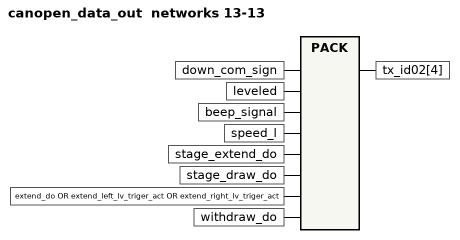
[picture p96: canopen_data_out (FBD) networks 13-13]
_FBD_ (* Function Block Diagram *)
NETWORK 1
	PACK(front_left_urt_ex_check, front_right_urt_ex_check, back_left_urt_ex_check, back_right_urt_ex_check, front_left_urt_drb_check, front_right_urt_drb_check, back_left_urt_drb_check, back_right_urt_drb_check) => tx_id01[0]
NETWORK 2
	PACK(front_left_Lv_ex_check, front_right_Lv_ex_check, back_left_Lv_ex_check, back_right_Lv_ex_check, front_left_Lv_drb_check, front_right_Lv_drb_check, back_left_Lv_drb_check, back_right_Lv_drb_check) => tx_id01[1]
NETWORK 3
	PACK(engine_run, engine_stop, accelerate_sb, decelerate_sb, down_force, tt_forcexx, standby_pump_check, water_pump_run_sb) => tx_id01[2]
NETWORK 4
	PACK(auto_manu_choice, left_side_choice, right_side_choice, level_extend_triger_left, level_extend_triger_right, auto_extend_triger_left OR auto_extend_triger_right, auto_drawback_triger_left OR auto_drawback_triger_right, remote_switch_leg) => tx_id01[3]
NETWORK 5
	PACK(FALSE, FALSE, FALSE, FALSE, FALSE, FALSE, FALSE, FALSE) => tx_id01[4]
NETWORK 6
	PACK(FALSE, FALSE, FALSE, FALSE, FALSE, FALSE, FALSE, FALSE) => tx_id01[5]
NETWORK 7
	PACK(arm_to_station, water_pump_check, left_groud_check1, left_groud_check2, oil_pump_check, FALSE, FALSE, FALSE) => tx_id01[6]
NETWORK 8
	PACK(FALSE, FALSE, FALSE, FALSE, FALSE, FALSE, FALSE, FALSE) => tx_id01[7]
NETWORK 9
	PACK(left_front_lv_ex_valve, right_front_lv_ex_valve, left_back_lv_ex_valve, right_back_lv_ex_valve, left_front_lv_drb_valve, right_front_lv_drb_valve, left_back_lv_drb_valve, right_back_lv_drb_valve) => tx_id02[0]
NETWORK 10
	PACK(enginer_run_ctl, enginer_stop_ctl, enginer_acc_ctl, enginer_dec_ctl, water_pump_ctl, up_valve_ctl, down_valve_ctl, over_level_sign) => tx_id02[1]
NETWORK 11
	PACK(triger_left_grd_sign, under_reset_ctl, standby_oil_pump, triger_flash, triger_no_drawback_sign, leveled_sign, alarmer_horn, FALSE) => tx_id02[2]
NETWORK 12
	PACK(FALSE, FALSE, FALSE, FALSE, FALSE, FALSE, FALSE, FALSE) => tx_id02[3]
NETWORK 13
	PACK(down_com_sign, leveled, beep_signal, speed_l, stage_extend_do, stage_draw_do, extend_do OR extend_left_lv_triger_act OR extend_right_lv_triger_act, withdraw_do) => tx_id02[4]
_END_FBD_
(* the same logic as Structured Text *)
(* Network 1 *)
tx_id01[0] := PACK(front_left_urt_ex_check, front_right_urt_ex_check, back_left_urt_ex_check, back_right_urt_ex_check, front_left_urt_drb_check, front_right_urt_drb_check, back_left_urt_drb_check, back_right_urt_drb_check);
(* Network 2 *)
tx_id01[1] := PACK(front_left_Lv_ex_check, front_right_Lv_ex_check, back_left_Lv_ex_check, back_right_Lv_ex_check, front_left_Lv_drb_check, front_right_Lv_drb_check, back_left_Lv_drb_check, back_right_Lv_drb_check);
(* Network 3 *)
tx_id01[2] := PACK(engine_run, engine_stop, accelerate_sb, decelerate_sb, down_force, tt_forcexx, standby_pump_check, water_pump_run_sb);
(* Network 4 *)
tx_id01[3] := PACK(auto_manu_choice, left_side_choice, right_side_choice, level_extend_triger_left, level_extend_triger_right, auto_extend_triger_left OR auto_extend_triger_right, auto_drawback_triger_left OR auto_drawback_triger_right, remote_switch_leg);
(* Network 5 *)
tx_id01[4] := PACK(FALSE, FALSE, FALSE, FALSE, FALSE, FALSE, FALSE, FALSE);
(* Network 6 *)
tx_id01[5] := PACK(FALSE, FALSE, FALSE, FALSE, FALSE, FALSE, FALSE, FALSE);
(* Network 7 *)
tx_id01[6] := PACK(arm_to_station, water_pump_check, left_groud_check1, left_groud_check2, oil_pump_check, FALSE, FALSE, FALSE);
(* Network 8 *)
tx_id01[7] := PACK(FALSE, FALSE, FALSE, FALSE, FALSE, FALSE, FALSE, FALSE);
(* Network 9 *)
tx_id02[0] := PACK(left_front_lv_ex_valve, right_front_lv_ex_valve, left_back_lv_ex_valve, right_back_lv_ex_valve, left_front_lv_drb_valve, right_front_lv_drb_valve, left_back_lv_drb_valve, right_back_lv_drb_valve);
(* Network 10 *)
tx_id02[1] := PACK(enginer_run_ctl, enginer_stop_ctl, enginer_acc_ctl, enginer_dec_ctl, water_pump_ctl, up_valve_ctl, down_valve_ctl, over_level_sign);
(* Network 11 *)
tx_id02[2] := PACK(triger_left_grd_sign, under_reset_ctl, standby_oil_pump, triger_flash, triger_no_drawback_sign, leveled_sign, alarmer_horn, FALSE);
(* Network 12 *)
tx_id02[3] := PACK(FALSE, FALSE, FALSE, FALSE, FALSE, FALSE, FALSE, FALSE);
(* Network 13 *)
tx_id02[4] := PACK(down_com_sign, leveled, beep_signal, speed_l, stage_extend_do, stage_draw_do, extend_do OR extend_left_lv_triger_act OR extend_right_lv_triger_act, withdraw_do);
END_PROGRAM

(* POU CANOPEN_DATA/digit_data_in, FBD *)
PROGRAM digit_data_in
VAR

	UNPACK1		: UNPACK;
	UNPACK2		: UNPACK;
	UNPACK3		: UNPACK;
	UNPACK4		: UNPACK;
	UNPACK5		: UNPACK;
	UNPACK6		: UNPACK;
	UNPACK7		: UNPACK;
	UNPACK8		: UNPACK;
	UNPACK9		: UNPACK;
	UNPACK10	: UNPACK;
	UNPACK11	: UNPACK;

END_VAR
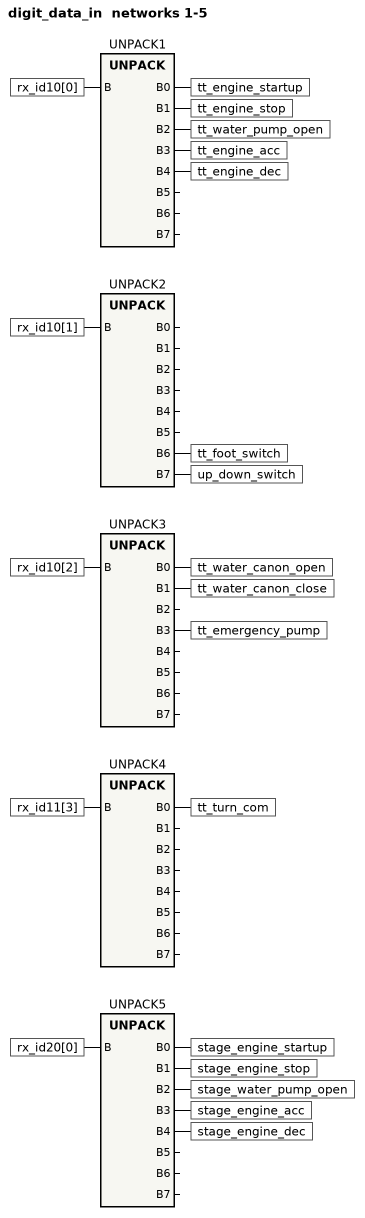
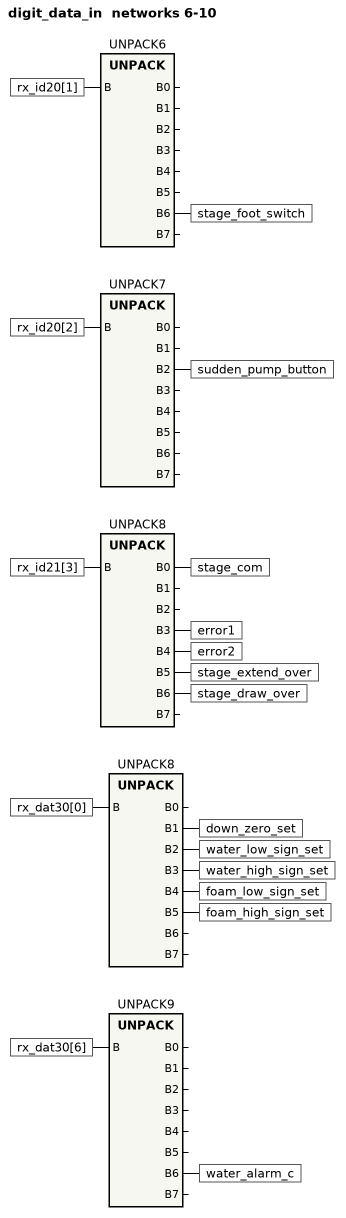
_FBD_ (* Function Block Diagram *)
NETWORK 1
	UNPACK1:UNPACK(B: rx_id10[0], B1 => tt_engine_stop, B2 => tt_water_pump_open, B3 => tt_engine_acc, B4 => tt_engine_dec) => tt_engine_startup
NETWORK 2
	UNPACK2:UNPACK(B: rx_id10[1], B6 => tt_foot_switch, B7 => up_down_switch)
NETWORK 3
	UNPACK3:UNPACK(B: rx_id10[2], B1 => tt_water_canon_close, B3 => tt_emergency_pump) => tt_water_canon_open
NETWORK 4
	UNPACK4:UNPACK(B: rx_id11[3]) => tt_turn_com
NETWORK 5
	UNPACK5:UNPACK(B: rx_id20[0], B1 => stage_engine_stop, B2 => stage_water_pump_open, B3 => stage_engine_acc, B4 => stage_engine_dec) => stage_engine_startup
NETWORK 6
	UNPACK6:UNPACK(B: rx_id20[1], B6 => stage_foot_switch)
NETWORK 7
	UNPACK7:UNPACK(B: rx_id20[2], B2 => sudden_pump_button)
NETWORK 8
	UNPACK8:UNPACK(B: rx_id21[3], B3 => error1, B4 => error2, B5 => stage_extend_over, B6 => stage_draw_over) => stage_com
NETWORK 9
	UNPACK8:UNPACK(B: rx_dat30[0], B1 => down_zero_set, B2 => water_low_sign_set, B3 => water_high_sign_set, B4 => foam_low_sign_set, B5 => foam_high_sign_set)
NETWORK 10
	UNPACK9:UNPACK(B: rx_dat30[6], B6 => water_alarm_c)
_END_FBD_
(* the same logic as Structured Text *)
(* Network 1 *)
UNPACK1(B := rx_id10[0]);
tt_engine_stop := UNPACK1.B1;
tt_water_pump_open := UNPACK1.B2;
tt_engine_acc := UNPACK1.B3;
tt_engine_dec := UNPACK1.B4;
tt_engine_startup := UNPACK1.B0;
(* Network 2 *)
UNPACK2(B := rx_id10[1]);
tt_foot_switch := UNPACK2.B6;
up_down_switch := UNPACK2.B7;
(* Network 3 *)
UNPACK3(B := rx_id10[2]);
tt_water_canon_close := UNPACK3.B1;
tt_emergency_pump := UNPACK3.B3;
tt_water_canon_open := UNPACK3.B0;
(* Network 4 *)
UNPACK4(B := rx_id11[3]);
tt_turn_com := UNPACK4.B0;
(* Network 5 *)
UNPACK5(B := rx_id20[0]);
stage_engine_stop := UNPACK5.B1;
stage_water_pump_open := UNPACK5.B2;
stage_engine_acc := UNPACK5.B3;
stage_engine_dec := UNPACK5.B4;
stage_engine_startup := UNPACK5.B0;
(* Network 6 *)
UNPACK6(B := rx_id20[1]);
stage_foot_switch := UNPACK6.B6;
(* Network 7 *)
UNPACK7(B := rx_id20[2]);
sudden_pump_button := UNPACK7.B2;
(* Network 8 *)
UNPACK8(B := rx_id21[3]);
error1 := UNPACK8.B3;
error2 := UNPACK8.B4;
stage_extend_over := UNPACK8.B5;
stage_draw_over := UNPACK8.B6;
stage_com := UNPACK8.B0;
(* Network 9 *)
UNPACK8(B := rx_dat30[0]);
down_zero_set := UNPACK8.B1;
water_low_sign_set := UNPACK8.B2;
water_high_sign_set := UNPACK8.B3;
foam_low_sign_set := UNPACK8.B4;
foam_high_sign_set := UNPACK8.B5;
(* Network 10 *)
UNPACK9(B := rx_dat30[6]);
water_alarm_c := UNPACK9.B6;
END_PROGRAM

(* POU alarm_text/ALARM_TEXT, FBD *)
PROGRAM ALARM_TEXT
VAR

END_VAR
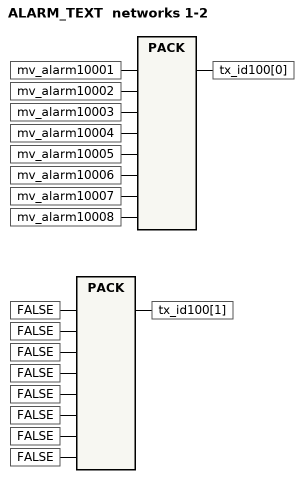
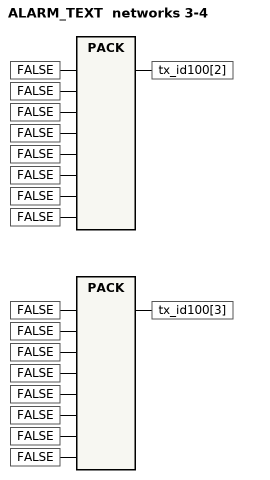
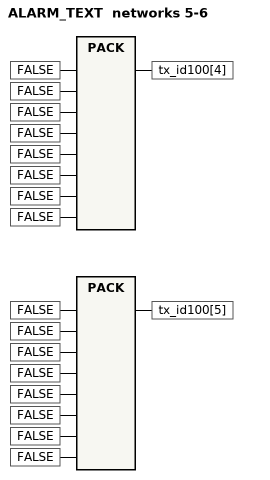
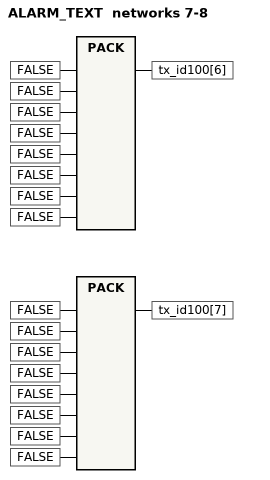
_FBD_ (* Function Block Diagram *)
NETWORK 1
	PACK(mv_alarm10001, mv_alarm10002, mv_alarm10003, mv_alarm10004, mv_alarm10005, mv_alarm10006, mv_alarm10007, mv_alarm10008) => tx_id100[0]
NETWORK 2
	PACK(FALSE, FALSE, FALSE, FALSE, FALSE, FALSE, FALSE, FALSE) => tx_id100[1]
NETWORK 3
	PACK(FALSE, FALSE, FALSE, FALSE, FALSE, FALSE, FALSE, FALSE) => tx_id100[2]
NETWORK 4
	PACK(FALSE, FALSE, FALSE, FALSE, FALSE, FALSE, FALSE, FALSE) => tx_id100[3]
NETWORK 5
	PACK(FALSE, FALSE, FALSE, FALSE, FALSE, FALSE, FALSE, FALSE) => tx_id100[4]
NETWORK 6
	PACK(FALSE, FALSE, FALSE, FALSE, FALSE, FALSE, FALSE, FALSE) => tx_id100[5]
NETWORK 7
	PACK(FALSE, FALSE, FALSE, FALSE, FALSE, FALSE, FALSE, FALSE) => tx_id100[6]
NETWORK 8
	PACK(FALSE, FALSE, FALSE, FALSE, FALSE, FALSE, FALSE, FALSE) => tx_id100[7]
_END_FBD_
(* the same logic as Structured Text *)
(* Network 1 *)
tx_id100[0] := PACK(mv_alarm10001, mv_alarm10002, mv_alarm10003, mv_alarm10004, mv_alarm10005, mv_alarm10006, mv_alarm10007, mv_alarm10008);
(* Network 2 *)
tx_id100[1] := PACK(FALSE, FALSE, FALSE, FALSE, FALSE, FALSE, FALSE, FALSE);
(* Network 3 *)
tx_id100[2] := PACK(FALSE, FALSE, FALSE, FALSE, FALSE, FALSE, FALSE, FALSE);
(* Network 4 *)
tx_id100[3] := PACK(FALSE, FALSE, FALSE, FALSE, FALSE, FALSE, FALSE, FALSE);
(* Network 5 *)
tx_id100[4] := PACK(FALSE, FALSE, FALSE, FALSE, FALSE, FALSE, FALSE, FALSE);
(* Network 6 *)
tx_id100[5] := PACK(FALSE, FALSE, FALSE, FALSE, FALSE, FALSE, FALSE, FALSE);
(* Network 7 *)
tx_id100[6] := PACK(FALSE, FALSE, FALSE, FALSE, FALSE, FALSE, FALSE, FALSE);
(* Network 8 *)
tx_id100[7] := PACK(FALSE, FALSE, FALSE, FALSE, FALSE, FALSE, FALSE, FALSE);
END_PROGRAM

(* POU PLC_CYCLE, ST *)
PROGRAM PLC_CYCLE
VAR
	old_cycle: DWORD;
	TIMER_READ_US1: TIMER_READ_US;
	cycle: DWORD;
	init: BOOL:=TRUE;
END_VAR
VAR_OUTPUT
	cycletime_us: DWORD;
	max_cycle_us: DWORD;
END_VAR

VAR_INPUT
	reset_max_cycletime: BOOL;
END_VAR
	TIMER_READ_US1(TIME_US=>cycle );
	cycletime_us:=cycle-old_cycle;
	old_cycle:=cycle;

	IF max_cycle_us<cycletime_us AND NOT init THEN
		max_cycle_us:=cycletime_us;
	END_IF;

	IF reset_max_cycletime THEN
		max_cycle_us:=0;
	END_IF;

	init:=FALSE;
END_PROGRAM

(* POU CAN_OPEN/CANOPEN, FBD *)
PROGRAM CANOPEN
VAR
	Status: CAN1_MASTER_STATUS;


	LedStatus: BOOL:= TRUE;
	StartAllNodes: BOOL:= TRUE;
	ClearRxOverflowFlag: BOOL;
	ClearRxBuffer: BOOL;
	ClearTxOverflowFlag: BOOL;
	ClearTxBuffer: BOOL;
	ClearOdChanged: BOOL;
	ClearErrorControl: BOOL;
	ResetAllNodes: BOOL;

	NodeStateSlavesArray: ARRAY [0..MAX_NODEINDEX] OF CAN1_NODE_STATE;
	EmergencyObjectSlavesArray: ARRAY[0..MAX_NODEINDEX] OF CAN1_EMERGENCY_MESSAGE;
	my_node_id: BYTE;
	my_baudrate: WORD;
	my_node_state: INT;
	Sync: BOOL;
	RxOverflow: BOOL;
	TxOverflow: BOOL;
	OdChanged: BOOL;
	GuardHeartbeatErrorArray: ARRAY[0..7] OF BYTE;
	GetEmergency: CAN1_EMERGENCY_MESSAGE;



	start2: BOOL;
	Emcy_handler: CAN1_MASTER_EMCY_HANDLER;
	reset_emcy: BOOL;
END_VAR
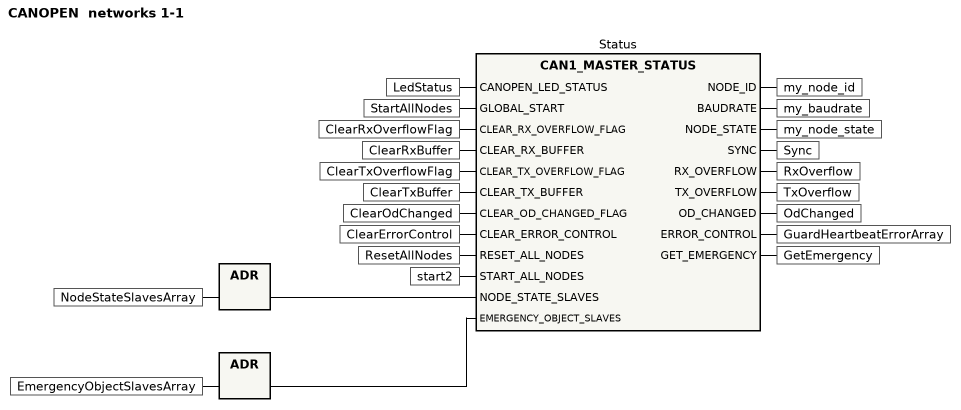
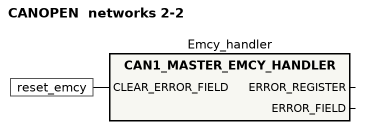
_FBD_ (* Function Block Diagram *)
NETWORK 1
	Status:CAN1_MASTER_STATUS(CANOPEN_LED_STATUS: LedStatus, GLOBAL_START: StartAllNodes, CLEAR_RX_OVERFLOW_FLAG: ClearRxOverflowFlag, CLEAR_RX_BUFFER: ClearRxBuffer, CLEAR_TX_OVERFLOW_FLAG: ClearTxOverflowFlag, CLEAR_TX_BUFFER: ClearTxBuffer, CLEAR_OD_CHANGED_FLAG: ClearOdChanged, CLEAR_ERROR_CONTROL: ClearErrorControl, RESET_ALL_NODES: ResetAllNodes, START_ALL_NODES: start2, NODE_STATE_SLAVES: ADR(NodeStateSlavesArray), EMERGENCY_OBJECT_SLAVES: ADR(EmergencyObjectSlavesArray), BAUDRATE => my_baudrate, NODE_STATE => my_node_state, SYNC => Sync, RX_OVERFLOW => RxOverflow, TX_OVERFLOW => TxOverflow, OD_CHANGED => OdChanged, ERROR_CONTROL => GuardHeartbeatErrorArray, GET_EMERGENCY => GetEmergency) => my_node_id
NETWORK 2
	Emcy_handler:CAN1_MASTER_EMCY_HANDLER(CLEAR_ERROR_FIELD: reset_emcy)
_END_FBD_
(* the same logic as Structured Text *)
(* Network 1 *)
Status(CANOPEN_LED_STATUS := LedStatus, GLOBAL_START := StartAllNodes, CLEAR_RX_OVERFLOW_FLAG := ClearRxOverflowFlag, CLEAR_RX_BUFFER := ClearRxBuffer, CLEAR_TX_OVERFLOW_FLAG := ClearTxOverflowFlag, CLEAR_TX_BUFFER := ClearTxBuffer, CLEAR_OD_CHANGED_FLAG := ClearOdChanged, CLEAR_ERROR_CONTROL := ClearErrorControl, RESET_ALL_NODES := ResetAllNodes, START_ALL_NODES := start2, NODE_STATE_SLAVES := ADR(NodeStateSlavesArray), EMERGENCY_OBJECT_SLAVES := ADR(EmergencyObjectSlavesArray));
my_baudrate := Status.BAUDRATE;
my_node_state := Status.NODE_STATE;
Sync := Status.SYNC;
RxOverflow := Status.RX_OVERFLOW;
TxOverflow := Status.TX_OVERFLOW;
OdChanged := Status.OD_CHANGED;
GuardHeartbeatErrorArray := Status.ERROR_CONTROL;
GetEmergency := Status.GET_EMERGENCY;
my_node_id := Status.NODE_ID;
(* Network 2 *)
Emcy_handler(CLEAR_ERROR_FIELD := reset_emcy);
END_PROGRAM

(* POU CANOPEN_DATA/CANOPEN_DATA_OUT2, FBD *)
PROGRAM CANOPEN_DATA_OUT2
VAR

END_VAR
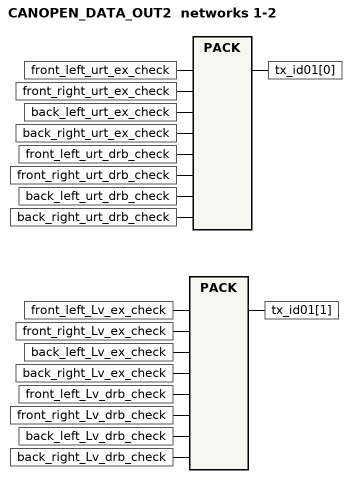
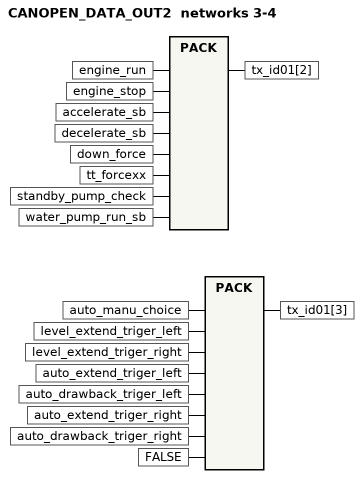
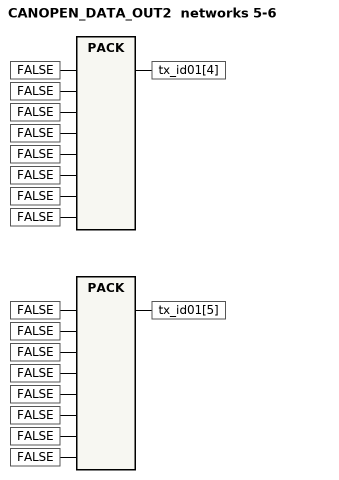
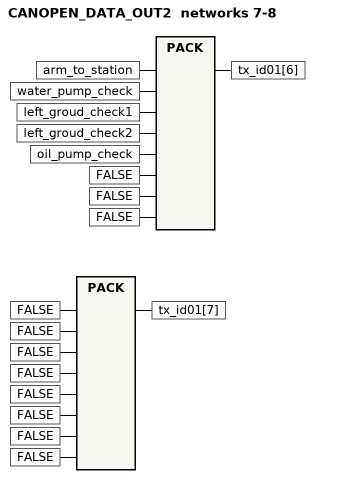
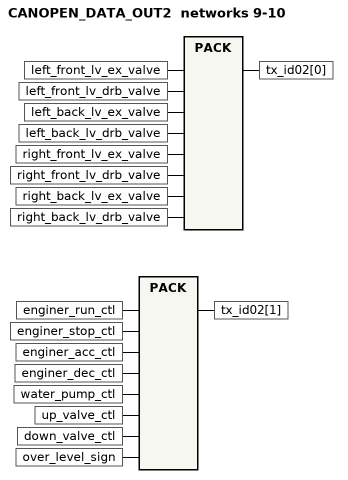
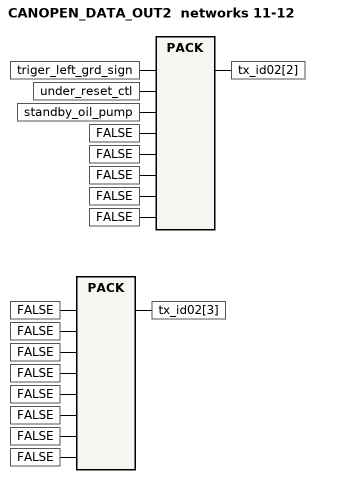
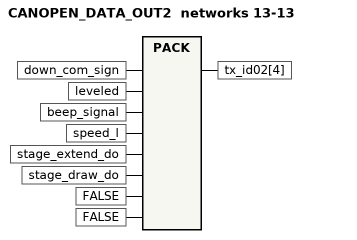
_FBD_ (* Function Block Diagram *)
NETWORK 1
	PACK(front_left_urt_ex_check, front_right_urt_ex_check, back_left_urt_ex_check, back_right_urt_ex_check, front_left_urt_drb_check, front_right_urt_drb_check, back_left_urt_drb_check, back_right_urt_drb_check) => tx_id01[0]
NETWORK 2
	PACK(front_left_Lv_ex_check, front_right_Lv_ex_check, back_left_Lv_ex_check, back_right_Lv_ex_check, front_left_Lv_drb_check, front_right_Lv_drb_check, back_left_Lv_drb_check, back_right_Lv_drb_check) => tx_id01[1]
NETWORK 3
	PACK(engine_run, engine_stop, accelerate_sb, decelerate_sb, down_force, tt_forcexx, standby_pump_check, water_pump_run_sb) => tx_id01[2]
NETWORK 4
	PACK(auto_manu_choice, level_extend_triger_left, level_extend_triger_right, auto_extend_triger_left, auto_drawback_triger_left, auto_extend_triger_right, auto_drawback_triger_right, FALSE) => tx_id01[3]
NETWORK 5
	PACK(FALSE, FALSE, FALSE, FALSE, FALSE, FALSE, FALSE, FALSE) => tx_id01[4]
NETWORK 6
	PACK(FALSE, FALSE, FALSE, FALSE, FALSE, FALSE, FALSE, FALSE) => tx_id01[5]
NETWORK 7
	PACK(arm_to_station, water_pump_check, left_groud_check1, left_groud_check2, oil_pump_check, FALSE, FALSE, FALSE) => tx_id01[6]
NETWORK 8
	PACK(FALSE, FALSE, FALSE, FALSE, FALSE, FALSE, FALSE, FALSE) => tx_id01[7]
NETWORK 9
	PACK(left_front_lv_ex_valve, left_front_lv_drb_valve, left_back_lv_ex_valve, left_back_lv_drb_valve, right_front_lv_ex_valve, right_front_lv_drb_valve, right_back_lv_ex_valve, right_back_lv_drb_valve) => tx_id02[0]
NETWORK 10
	PACK(enginer_run_ctl, enginer_stop_ctl, enginer_acc_ctl, enginer_dec_ctl, water_pump_ctl, up_valve_ctl, down_valve_ctl, over_level_sign) => tx_id02[1]
NETWORK 11
	PACK(triger_left_grd_sign, under_reset_ctl, standby_oil_pump, FALSE, FALSE, FALSE, FALSE, FALSE) => tx_id02[2]
NETWORK 12
	PACK(FALSE, FALSE, FALSE, FALSE, FALSE, FALSE, FALSE, FALSE) => tx_id02[3]
NETWORK 13
	PACK(down_com_sign, leveled, beep_signal, speed_l, stage_extend_do, stage_draw_do, FALSE, FALSE) => tx_id02[4]
_END_FBD_
(* the same logic as Structured Text *)
(* Network 1 *)
tx_id01[0] := PACK(front_left_urt_ex_check, front_right_urt_ex_check, back_left_urt_ex_check, back_right_urt_ex_check, front_left_urt_drb_check, front_right_urt_drb_check, back_left_urt_drb_check, back_right_urt_drb_check);
(* Network 2 *)
tx_id01[1] := PACK(front_left_Lv_ex_check, front_right_Lv_ex_check, back_left_Lv_ex_check, back_right_Lv_ex_check, front_left_Lv_drb_check, front_right_Lv_drb_check, back_left_Lv_drb_check, back_right_Lv_drb_check);
(* Network 3 *)
tx_id01[2] := PACK(engine_run, engine_stop, accelerate_sb, decelerate_sb, down_force, tt_forcexx, standby_pump_check, water_pump_run_sb);
(* Network 4 *)
tx_id01[3] := PACK(auto_manu_choice, level_extend_triger_left, level_extend_triger_right, auto_extend_triger_left, auto_drawback_triger_left, auto_extend_triger_right, auto_drawback_triger_right, FALSE);
(* Network 5 *)
tx_id01[4] := PACK(FALSE, FALSE, FALSE, FALSE, FALSE, FALSE, FALSE, FALSE);
(* Network 6 *)
tx_id01[5] := PACK(FALSE, FALSE, FALSE, FALSE, FALSE, FALSE, FALSE, FALSE);
(* Network 7 *)
tx_id01[6] := PACK(arm_to_station, water_pump_check, left_groud_check1, left_groud_check2, oil_pump_check, FALSE, FALSE, FALSE);
(* Network 8 *)
tx_id01[7] := PACK(FALSE, FALSE, FALSE, FALSE, FALSE, FALSE, FALSE, FALSE);
(* Network 9 *)
tx_id02[0] := PACK(left_front_lv_ex_valve, left_front_lv_drb_valve, left_back_lv_ex_valve, left_back_lv_drb_valve, right_front_lv_ex_valve, right_front_lv_drb_valve, right_back_lv_ex_valve, right_back_lv_drb_valve);
(* Network 10 *)
tx_id02[1] := PACK(enginer_run_ctl, enginer_stop_ctl, enginer_acc_ctl, enginer_dec_ctl, water_pump_ctl, up_valve_ctl, down_valve_ctl, over_level_sign);
(* Network 11 *)
tx_id02[2] := PACK(triger_left_grd_sign, under_reset_ctl, standby_oil_pump, FALSE, FALSE, FALSE, FALSE, FALSE);
(* Network 12 *)
tx_id02[3] := PACK(FALSE, FALSE, FALSE, FALSE, FALSE, FALSE, FALSE, FALSE);
(* Network 13 *)
tx_id02[4] := PACK(down_com_sign, leveled, beep_signal, speed_l, stage_extend_do, stage_draw_do, FALSE, FALSE);
END_PROGRAM

(* POU PDM_COM_LAYER2/PLC_TO_PDM, ST *)
PROGRAM PLC_TO_PDM
VAR_INPUT

	ENABLE: BOOL;
	INIT: BOOL;
	TRANSMIT_TIME:TIME;	(*if transmit time=0, both id's transmit asynchron*)
	GUARD_TIME:TIME;
	TX_ID1: WORD;
	TX_ID2: WORD;
	RX_ID1:WORD;
	RX_ID2:WORD;

END_VAR
VAR_OUTPUT

	ERROR_COMUNICATION: BOOL;

END_VAR
VAR

	Send1: CAN1_TRANSMIT;
	Send2: CAN1_TRANSMIT;
	Rec1: CAN1_RECEIVE;
	Rec2: CAN1_RECEIVE;
	async_send1: BOOL;
	async_send2: BOOL;
	clock: BOOL;
	VarDword:DWORD;
	VarWord:WORD;
	T1: TON;
	one: BOOL;
	rec_ok: BOOL;

	Fl_rec_ok: R_TRIG;
	T_guard_on: TON;
	T_guard_off: TON;
	guard_clock_on: BOOL;
	guard_clock_off: BOOL;


	page_old: WORD;
	message_old: BYTE;
	message_group_old: BYTE;
	led_F_key_old: BYTE;
	led_control_key_old: BYTE;
	led_value_max_old: BYTE;
	led_value_night_old: BYTE;
	BacklightOld:BYTE;
	HandleOld:WORD;
	InputValueOld:DWORD;
	LengthOld:BYTE;
	ValueWord: WORD;

END_VAR
IF enable THEN
(****************Build a sync for transmit*************************)
	IF transmit_time< T#50ms THEN
		transmit_time:=T#50ms;
	END_IF;
	IF transmit_time=T#0ms THEN	(*if no transmit time set sync to 100ms*)
		transmit_time:=T#100ms;
	END_IF;
	T1(IN:=NOT T1.Q , PT:=transmit_time );
	clock:= T1.Q;

(*^^^^^^^^^^^^^^^^^^^^^^^^^^^^^^^^^^^^^^^^^^^^^^^^^^^^^^^^^^^^^^^^^^*)
(*************************Build the async for transmit*****************)
	IF page_old<>DESIRED_PAGE THEN
		page_old:=DESIRED_PAGE;
		async_send1:=TRUE;
	END_IF;
	IF message_old<>DESIRED_MESSAGE THEN
		message_old:=DESIRED_MESSAGE;
		async_send1:=TRUE;
	END_IF;
	IF message_group_old<>DESIRED_MESSAGE_GROUP THEN
		message_group_old:=DESIRED_MESSAGE_GROUP;
		async_send1:=TRUE;
	END_IF;
	IF led_F_key_old<>LED_F_KEYS THEN
		led_F_key_old:=LED_F_KEYS;
		async_send1:=TRUE;
	END_IF;
	IF led_control_key_old<>LED_C_KEYS THEN
		led_control_key_old:=LED_C_KEYS;
		async_send1:=TRUE;
	END_IF;
	IF led_value_max_old<>DESIRED_LEDVALUE_MAX THEN
		led_value_max_old:=DESIRED_LEDVALUE_MAX;
		async_send1:=TRUE;
	END_IF;
	IF led_value_night_old<>DESIRED_LEDVALUE_NIGHT THEN
		led_value_night_old:=DESIRED_LEDVALUE_NIGHT;
		async_send1:=TRUE;
	END_IF;
	IF BacklightOld<>DESIRED_BACKLIGHT THEN
		BacklightOld:=DESIRED_BACKLIGHT;
		async_send2:=TRUE;
	END_IF;
	IF HandleOld<>HANDLE_BACK THEN
		HandleOld:=HANDLE_BACK;
		async_send2:=TRUE;
	END_IF;
	IF InputValueOld<>INPUT_VALUE_BACK THEN
		InputValueOld:=INPUT_VALUE_BACK;
		async_send2:=TRUE;
	END_IF;
	IF LengthOld<>LENGHT_BACK THEN
		LengthOld:=LENGHT_BACK;
		async_send2:=TRUE;
	END_IF;


(*^^^^^^^^^^^^^^^^^^^^^^^^^^^^^^^^^^^^^^^^^^^^^^^^^^^^^^^^^^^^^^^^^^*)

(************Build the guarding toggle and send it with backlight*****************************)
	IF DESIRED_BACKLIGHT>100 THEN
		DESIRED_BACKLIGHT:=100;
	END_IF;

	IF clock THEN
		one := NOT one;
	END_IF;
	Send2.DATA[0]:=DESIRED_BACKLIGHT;
	IF one THEN
		Send2.DATA[0].7:= TRUE;
		ELSE
			Send2.DATA[0].7:=FALSE;
	END_IF;
(*^^^^^^^^^^^^^^^^^^^^^^^^^^^^^^^^^^^^^^^^^^^^^^^^^^^^^^^^^^^^^^^^^^*)

(********************copy data to transmit array*********************)

	Send1.DATA[0] := WORD_TO_BYTE(DESIRED_PAGE);
	VarWord := SHR(DESIRED_PAGE,8);
	Send1.DATA[1] := WORD_TO_BYTE(VarWord);
	Send1.DATA[2] := DESIRED_MESSAGE;
	Send1.DATA[3] := DESIRED_MESSAGE_GROUP;
	Send1.DATA[4] := LED_F_KEYS;
	Send1.DATA[5] := LED_C_KEYS;
	Send1.DATA[6] := DESIRED_LEDVALUE_MAX;
	Send1.DATA[7] := DESIRED_LEDVALUE_NIGHT;

	Send2.DATA[1] := Rec2.DATA[1];
	Send2.DATA[2] := Rec2.DATA[2];
	Send2.DATA[3] := Rec2.DATA[3];
	Send2.DATA[4] := Rec2.DATA[4];
	Send2.DATA[5] := Rec2.DATA[5];
	Send2.DATA[6] := Rec2.DATA[6];
	Send2.DATA[7]:=Rec2.DATA[7];

(*^^^^^^^^^^^^^^^^^^^^^^^^^^^^^^^^^^^^^^^^^^^^^^^^^^^^^^^^^^^^^^^^^^^^^^^^^^^^^^^^^^^^*)

(**************send data************************)
	Send1(ID:=tx_id1 , DLC:=8 , DATA:= , ENABLE:=clock  OR async_send1);

	Send2(ID:=tx_id2 , DLC:=8 , DATA:= , ENABLE:=clock OR async_send2);

	async_send1:=FALSE;
	async_send2:=FALSE;
(*^^^^^^^^^^^^^^^^^^^^^^^^^^^^^^^^^^^^^^^^^^^^^^^^^^^^^^^^^^^^^^^^^^^^^^^^^^^^^^^^^^^^*)

(**************receive data************************)
	Rec1(CONFIG:=init , CLEAR:=FALSE , ID:=rx_id1 );
	Rec2(CONFIG:=init , CLEAR:=FALSE , ID:=rx_id2 );

	(**************************check guarding**********************************)
	Fl_rec_ok(CLK:=Rec2.DATA[0].7 , Q=>rec_ok );

	T_guard_on(IN:=rec_ok , PT:=guard_time , Q=>guard_clock_on);
	T_guard_off(IN:=NOT rec_ok , PT:=guard_time , Q=>guard_clock_off);


	IF guard_clock_on OR guard_clock_off THEN
		error_comunication := TRUE;
		ELSE
			error_comunication := FALSE;
	END_IF;
	(*^^^^^^^^^^^^^^^^^^^^^^^^^^^^^^^^^^^^^^^^^^^^^^^^^^^^^^^^^^^^^^^^^^^^^^^^^^^^*)

	(***********************copy reveived data***********************************)
	PRESENT_PAGE :=Rec1.DATA[1];
	PRESENT_PAGE := SHL(PRESENT_PAGE,8) OR Rec1.DATA[0];
	PRESENT_MESSAGE := Rec1.DATA[2];
	PRESENT_MESSAGE_GROUP := Rec1.DATA[3];
	F_KEYS := Rec1.DATA[4];
	C_KEYS := Rec1.DATA[5];
	PRESENT_LEDVALUE_MAX := Rec1.DATA[6];
	PRESENT_LEDVALUE_NIGHT := Rec1.DATA[7];

	PRESENT_BACKLIGHT:= 16#7F AND Rec2.DATA[0];
	HANDLE:= Rec2.DATA[2];
	HANDLE:=SHL(HANDLE,8) OR Rec2.DATA[1];
	LENGHT:= Rec2.DATA[7];


	IF LENGHT<1 THEN
		LENGHT:=1;
	END_IF;
	IF LENGHT=3 OR LENGHT>4 THEN
		LENGHT:=4;
	END_IF;


	CASE LENGHT OF

		1:	INPUT_VALUE:=Rec2.DATA[3];

		2:	INPUT_VALUE:=Rec2.DATA[4];
			INPUT_VALUE:=SHL(INPUT_VALUE,8) OR Rec2.DATA[3];

		4:	INPUT_VALUE:=Rec2.DATA[6];
			INPUT_VALUE:=SHL(INPUT_VALUE,8) OR Rec2.DATA[5];
			INPUT_VALUE:=SHL(INPUT_VALUE,8) OR Rec2.DATA[4];
			INPUT_VALUE:=SHL(INPUT_VALUE,8) OR Rec2.DATA[3];

	END_CASE;

	(*^^^^^^^^^^^^^^^^^^^^^^^^^^^^^^^^^^^^^^^^^^^^^^^^^^^^^^^^^^^^^^^^^^^^^^^^^^^^*)

(*^^^^^^^^^^^^^^^^^^^^^^^^^^^^^^^^^^^^^^^^^^^^^^^^^^^^^^^^^^^^^^^^^^^^^^^^^^^^^^^^^^^^^^^^^^^^^^^^^^^^^^^^^^^^^^^^^^^^^^^^^^^^^^^^^^^^^^^^^^^^*)
END_IF;
END_PROGRAM

(* POU PDM_COM_LAYER2/TO_PDM, FBD *)
PROGRAM TO_PDM
VAR
	picture_new: BYTE;
	message_new: BYTE;
	m_group_new: BYTE;
	led_f_key: BYTE;
	led_c_key: BYTE;
	led_value_max: BYTE;
	led_value_night: BYTE;
	backlight: BYTE:=100;
	error_com: BOOL;
	picture_act: BYTE;
	message_act: BYTE;
	m_group_act: BYTE;
	led_f1: BOOL;
	led_f2: BOOL;
	led_f3: BOOL;
	led_f4: BOOL;
	led_f5: BOOL;
	led_f6: BOOL;
	led_esc: BOOL;
	led_up: BOOL;
	led_ok: BOOL;
	led_left: BOOL;
	led_down: BOOL;
	led_right: BOOL;
	led_night: BOOL;

	led_value_act: BYTE;
	led_value_night_act: BYTE;
	backlight_act: BYTE;
	F_key: UNPACK;
	f1: BOOL;
	f2: BOOL;
	f3: BOOL;
	f4: BOOL;
	f5: BOOL;
	f6: BOOL;
	C_key: UNPACK;
	k_esc: BOOL;
	k_up: BOOL;
	k_ok: BOOL;
	k_left: BOOL;
	k_down: BOOL;
	k_right: BOOL;

	led_night_act: BOOL;
	guard_time: TIME := T#500ms;
END_VAR
VAR_INPUT
	init: BOOL;
END_VAR
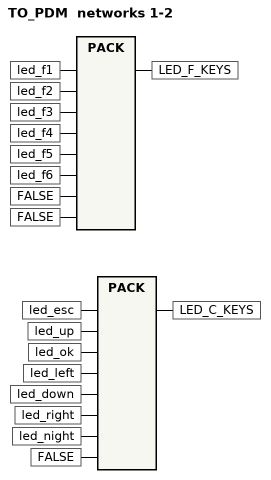
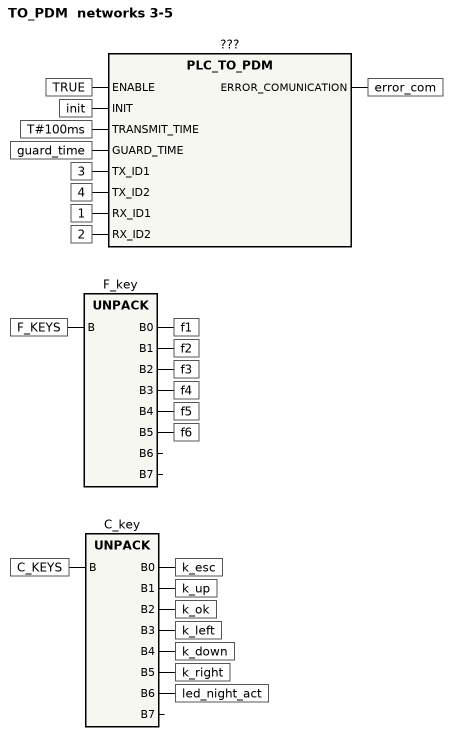
_FBD_ (* Function Block Diagram *)
NETWORK 1
	PACK(led_f1, led_f2, led_f3, led_f4, led_f5, led_f6, FALSE, FALSE) => LED_F_KEYS
NETWORK 2
	PACK(led_esc, led_up, led_ok, led_left, led_down, led_right, led_night, FALSE) => LED_C_KEYS
NETWORK 3
	???:PLC_TO_PDM(ENABLE: TRUE, INIT: init, TRANSMIT_TIME: T#100ms, GUARD_TIME: guard_time, TX_ID1: 3, TX_ID2: 4, RX_ID1: 1, RX_ID2: 2) => error_com
NETWORK 4
	F_key:UNPACK(B: F_KEYS, B1 => f2, B2 => f3, B3 => f4, B4 => f5, B5 => f6) => f1
NETWORK 5
	C_key:UNPACK(B: C_KEYS, B1 => k_up, B2 => k_ok, B3 => k_left, B4 => k_down, B5 => k_right, B6 => led_night_act) => k_esc
_END_FBD_
(* the same logic as Structured Text *)
(* Network 1 *)
LED_F_KEYS := PACK(led_f1, led_f2, led_f3, led_f4, led_f5, led_f6, FALSE, FALSE);
(* Network 2 *)
LED_C_KEYS := PACK(led_esc, led_up, led_ok, led_left, led_down, led_right, led_night, FALSE);
(* Network 3: see the listing above *)
(* Network 4 *)
F_key(B := F_KEYS);
f2 := F_key.B1;
f3 := F_key.B2;
f4 := F_key.B3;
f5 := F_key.B4;
f6 := F_key.B5;
f1 := F_key.B0;
(* Network 5 *)
C_key(B := C_KEYS);
k_up := C_key.B1;
k_ok := C_key.B2;
k_left := C_key.B3;
k_down := C_key.B4;
k_right := C_key.B5;
led_night_act := C_key.B6;
k_esc := C_key.B0;
END_PROGRAM
